Omron CX-Programmer project NewProject (CX-Programmer 9.61)

# PLC NewPLC1: CP1E N30

## Global symbols (name address type ; comment)
0.00 BOOL  ; PB1
100.00 BOOL  ; lampu
T000 BOOL  ; Timer1

## Program NewProgram1 (cyclic task 0)

### Section Section1

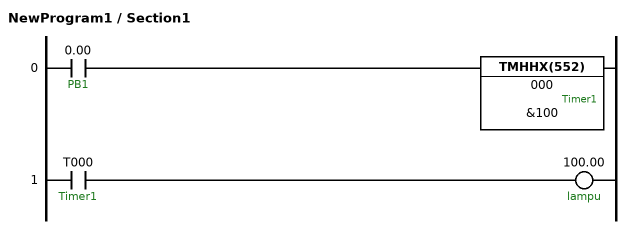
; rung 0
LD 0.00  ; PB1
TMHHX(552) 000 &100  ; Timer1
; rung 1
LD T000  ; Timer1
OUT 100.00  ; lampu

### Section END
; rung 0
END(001)